FUNCTION_BLOCK Test_TrimEx_HandlesEmptySubject EXTENDS T_UnitTestBase
VAR_INPUT
END_VAR
VAR_OUTPUT
END_VAR
VAR
    SubjectString : T_MaxString := '';
END_VAR

METHOD Init
VAR_INPUT
END_VAR
END_METHOD

{attribute 'analysis' := '-33'} // inhibit unused variable warning
METHOD RunTest
AssertEquals_STRING(Expected := '',
                    Actual   := F_Trim(str := SubjectString),
                    Message  := 'F_Trim(str := SubjectString)');

TestCompleted := TRUE;
END_METHOD

END_FUNCTION_BLOCK

(* stored: Version 1.1.0.1, ProductVersion 3.1.4024.12
   POU Test_TrimEx_HandlesEmptySubject: Id {d1276622-a662-0147-1776-f2ad3491e9d2}, SpecialFunc None
   Method Init: Id {f50a56f8-dd4e-0e6a-30a2-942459567b70}
   Method RunTest: Id {6fc06f30-baa2-062e-397f-5eaff5cce7db} *)
